(* Logix 5000 project; controller STAT 1756-L72 rev 20.12; software revision 20.04; part 24 of 34 *)
(* tags used below, declared in another part *)
   B3 : DINT[35];
   N9 : DINT[200];
   S : INT[164];
   T4 : TIMER[100];
   av310 : BOOL;
   av330 : BOOL;
   BITMW1 : BOOL;
   L4_R2_3_O : BOOL;
   S_AV310_V1_FC_C : BOOL;
   S_AV310_V1_FC_O : BOOL;
   S_AV310_V2_FC_C : BOOL;
   S_AV310_V2_FC_O : BOOL;
   S_AV330_V1_FC_C : BOOL;
   S_AV330_V1_FC_O : BOOL;
   S_AV330_V2_FC_C : BOOL;
   S_AV330_V2_FC_O : BOOL;
   stat_L1 : DINT[20];
   STAT_L3 : DINT[20];
(* LANCY, continued *)

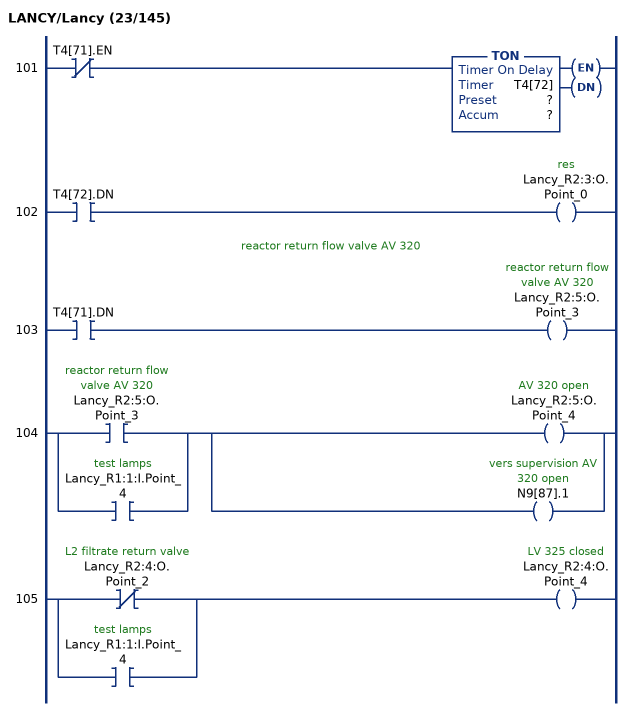
   101: XIO(T4[71].EN)TON(T4[72],?,?);
   102: XIC(T4[72].DN)OTE(Lancy_R2:3:O.Point_0);
   // reactor return flow valve AV 320
   103: XIC(T4[71].DN)OTE(Lancy_R2:5:O.Point_3);
   104: [XIC(Lancy_R2:5:O.Point_3) ,XIC(Lancy_R1:1:I.Point_4) ][OTE(Lancy_R2:5:O.Point_4) ,OTE(N9[87].1) ];
   105: [XIO(Lancy_R2:4:O.Point_2) ,XIC(Lancy_R1:1:I.Point_4) ]OTE(Lancy_R2:4:O.Point_4);
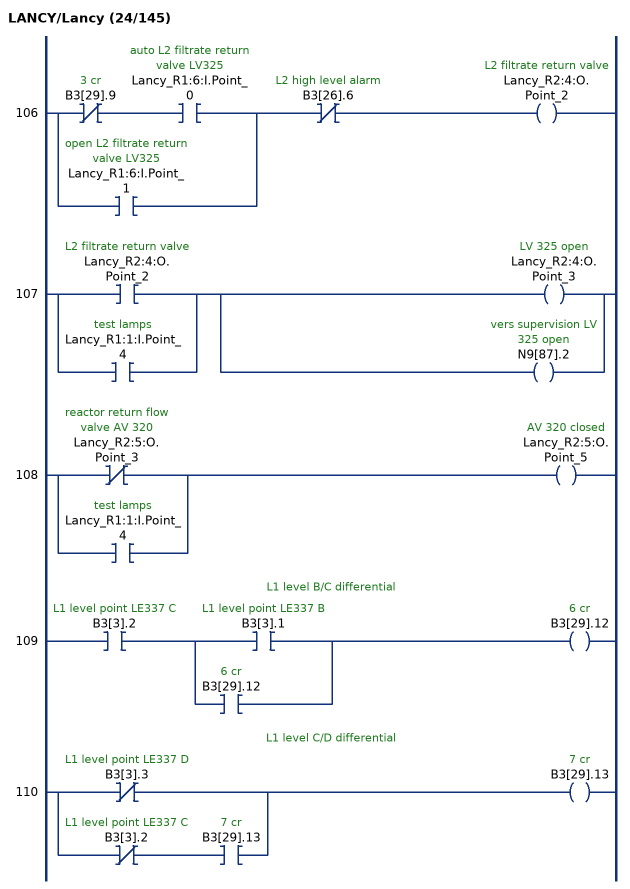
   106: [XIO(B3[29].9) XIC(Lancy_R1:6:I.Point_0) ,XIC(Lancy_R1:6:I.Point_1) ]XIO(B3[26].6)OTE(Lancy_R2:4:O.Point_2);
   107: [XIC(Lancy_R2:4:O.Point_2) ,XIC(Lancy_R1:1:I.Point_4) ][OTE(Lancy_R2:4:O.Point_3) ,OTE(N9[87].2) ];
   108: [XIO(Lancy_R2:5:O.Point_3) ,XIC(Lancy_R1:1:I.Point_4) ]OTE(Lancy_R2:5:O.Point_5);
   // L1 level B/C differential
   109: XIC(B3[3].2)[XIC(B3[3].1) ,XIC(B3[29].12) ]OTE(B3[29].12);
   // L1 level C/D differential
   110: [XIO(B3[3].3) ,XIO(B3[3].2) XIC(B3[29].13) ]OTE(B3[29].13);
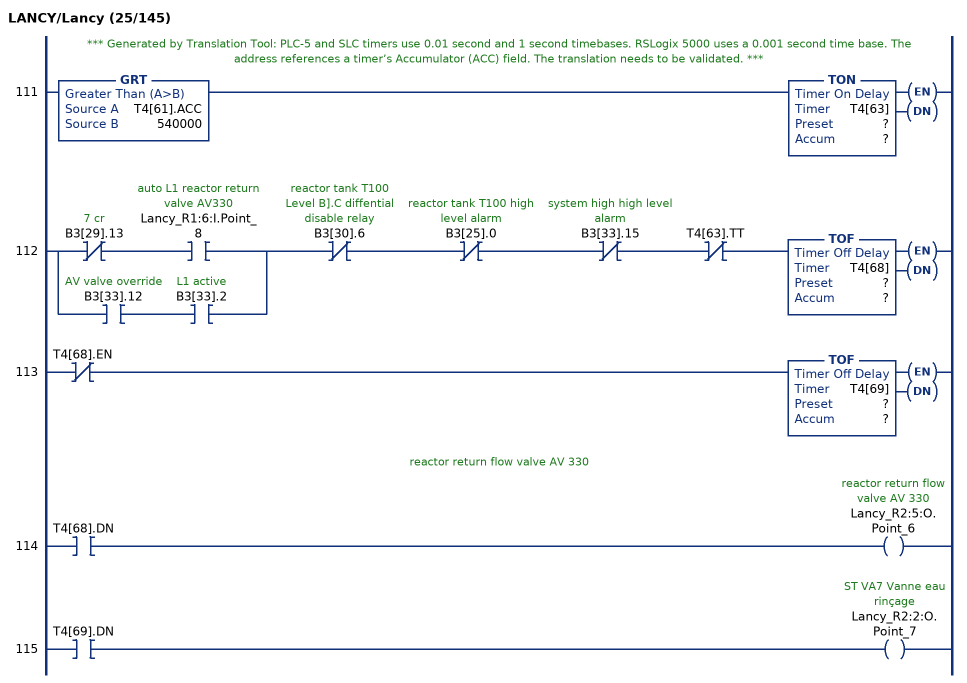
   // *** Generated by Translation Tool: PLC-5 and SLC timers use 0.01 second and 1 second timebases. RSLogix 5000 uses a 0.001 second time base. The address references a timer’s Accumulator (ACC) field. The translation needs to be validated. ***
   111: GRT(T4[61].ACC,540000)TON(T4[63],?,?);
   112: [XIO(B3[29].13) XIC(Lancy_R1:6:I.Point_8) ,XIC(B3[33].12) XIC(B3[33].2) ]XIO(B3[30].6)XIO(B3[25].0)XIO(B3[33].15)XIO(T4[63].TT)TOF(T4[68],?,?);
   113: XIO(T4[68].EN)TOF(T4[69],?,?);
   // reactor return flow valve AV 330
   114: XIC(T4[68].DN)OTE(Lancy_R2:5:O.Point_6);
   115: XIC(T4[69].DN)OTE(Lancy_R2:2:O.Point_7);
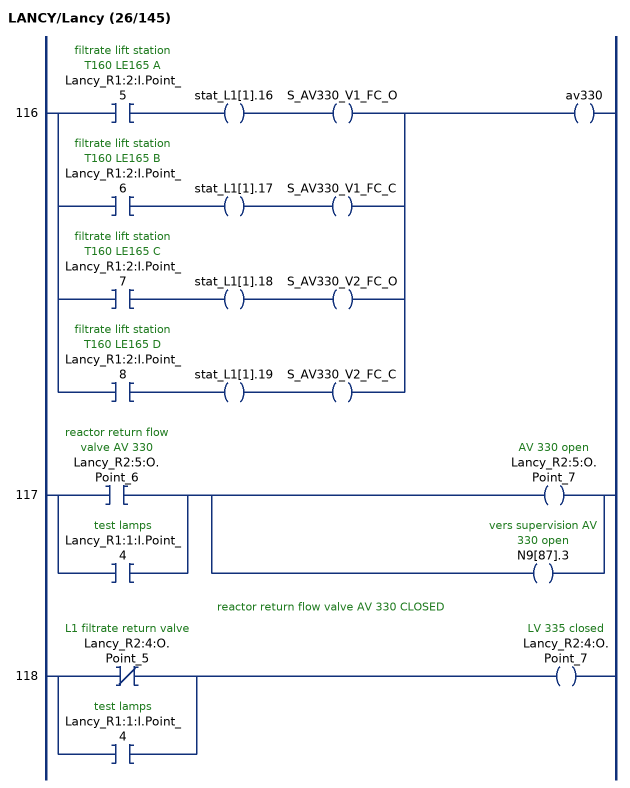
   116: [XIC(Lancy_R1:2:I.Point_5) OTE(stat_L1[1].16) OTE(S_AV330_V1_FC_O) ,XIC(Lancy_R1:2:I.Point_6) OTE(stat_L1[1].17) OTE(S_AV330_V1_FC_C) ,XIC(Lancy_R1:2:I.Point_7) OTE(stat_L1[1].18) OTE(S_AV330_V2_FC_O) ,XIC(Lancy_R1:2:I.Point_8) OTE(stat_L1[1].19) OTE(S_AV330_V2_FC_C) ]OTE(av330);
   117: [XIC(Lancy_R2:5:O.Point_6) ,XIC(Lancy_R1:1:I.Point_4) ][OTE(Lancy_R2:5:O.Point_7) ,OTE(N9[87].3) ];
   // reactor return flow valve AV 330 CLOSED
   118: [XIO(Lancy_R2:4:O.Point_5) ,XIC(Lancy_R1:1:I.Point_4) ]OTE(Lancy_R2:4:O.Point_7);
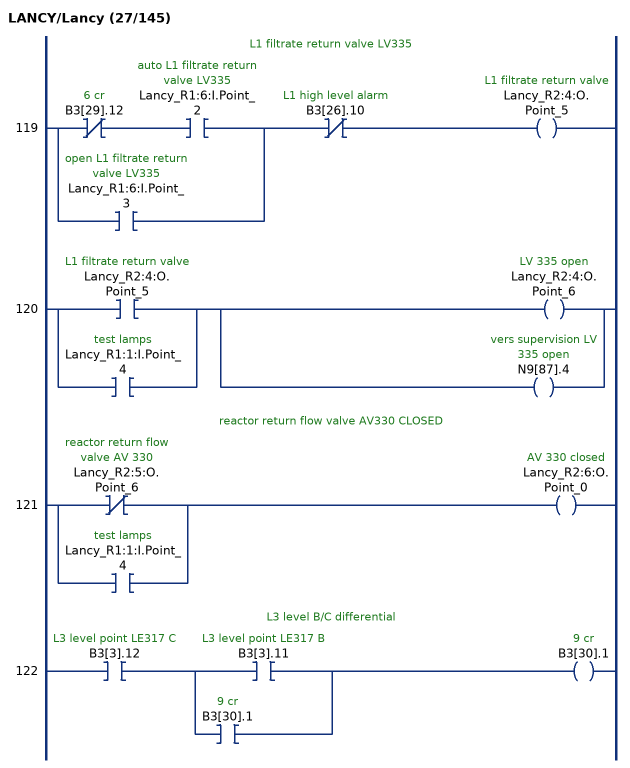
   // L1 filtrate return valve LV335
   119: [XIO(B3[29].12) XIC(Lancy_R1:6:I.Point_2) ,XIC(Lancy_R1:6:I.Point_3) ]XIO(B3[26].10)OTE(Lancy_R2:4:O.Point_5);
   120: [XIC(Lancy_R2:4:O.Point_5) ,XIC(Lancy_R1:1:I.Point_4) ][OTE(Lancy_R2:4:O.Point_6) ,OTE(N9[87].4) ];
   // reactor return flow valve AV330 CLOSED
   121: [XIO(Lancy_R2:5:O.Point_6) ,XIC(Lancy_R1:1:I.Point_4) ]OTE(Lancy_R2:6:O.Point_0);
   // L3 level B/C differential
   122: XIC(B3[3].12)[XIC(B3[3].11) ,XIC(B3[30].1) ]OTE(B3[30].1);
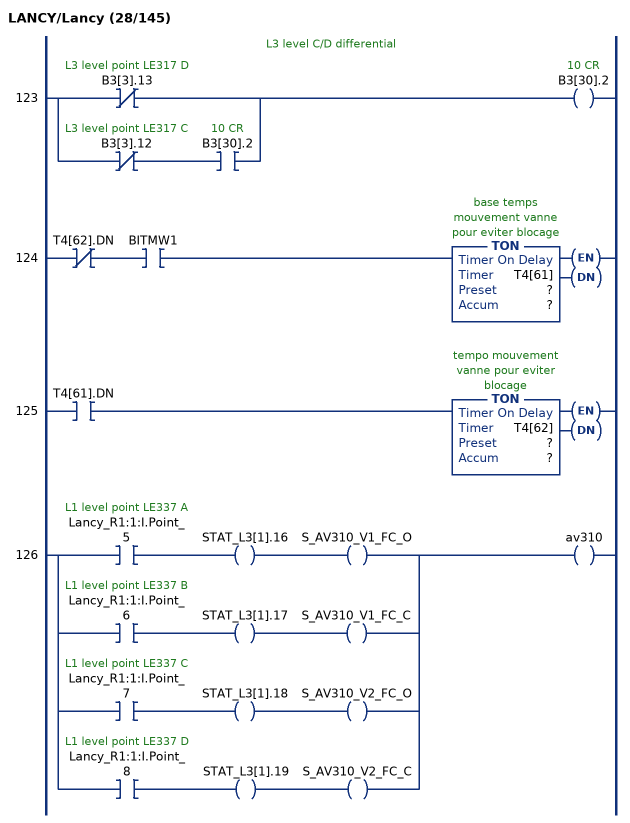
   // L3 level C/D differential
   123: [XIO(B3[3].13) ,XIO(B3[3].12) XIC(B3[30].2) ]OTE(B3[30].2);
   124: XIO(T4[62].DN)XIC(BITMW1)TON(T4[61],?,?);
   125: XIC(T4[61].DN)TON(T4[62],?,?);
   126: [XIC(Lancy_R1:1:I.Point_5) OTE(STAT_L3[1].16) OTE(S_AV310_V1_FC_O) ,XIC(Lancy_R1:1:I.Point_6) OTE(STAT_L3[1].17) OTE(S_AV310_V1_FC_C) ,XIC(Lancy_R1:1:I.Point_7) OTE(STAT_L3[1].18) OTE(S_AV310_V2_FC_O) ,XIC(Lancy_R1:1:I.Point_8) OTE(STAT_L3[1].19) OTE(S_AV310_V2_FC_C) ]OTE(av310);
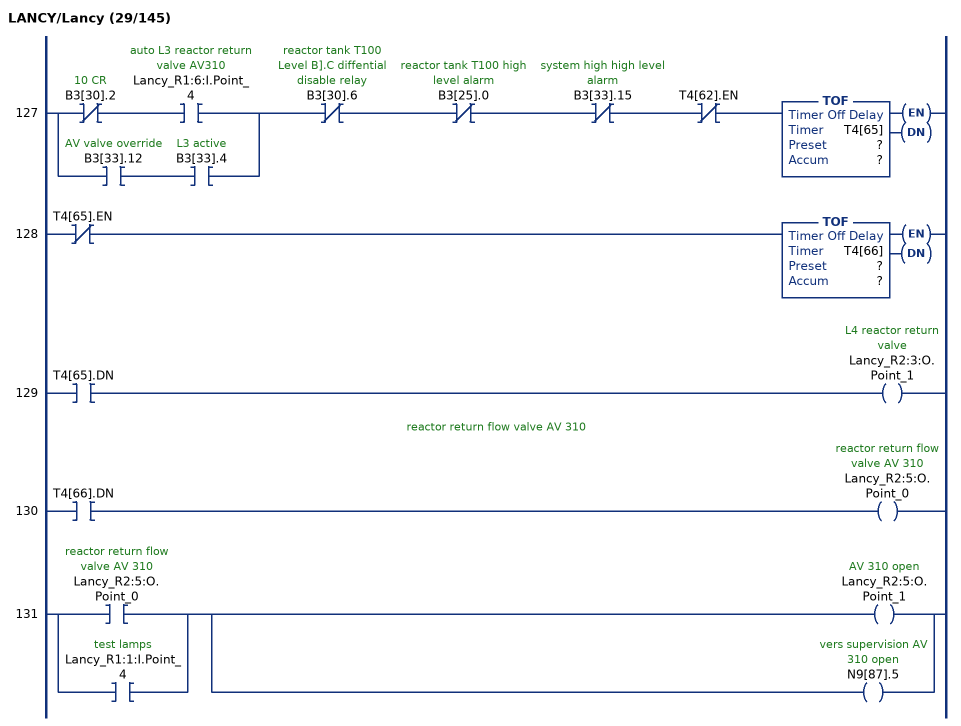
   127: [XIO(B3[30].2) XIC(Lancy_R1:6:I.Point_4) ,XIC(B3[33].12) XIC(B3[33].4) ]XIO(B3[30].6)XIO(B3[25].0)XIO(B3[33].15)XIO(T4[62].EN)TOF(T4[65],?,?);
   128: XIO(T4[65].EN)TOF(T4[66],?,?);
   129: XIC(T4[65].DN)OTE(Lancy_R2:3:O.Point_1);
   // reactor return flow valve AV 310
   130: XIC(T4[66].DN)OTE(Lancy_R2:5:O.Point_0);
   131: [XIC(Lancy_R2:5:O.Point_0) ,XIC(Lancy_R1:1:I.Point_4) ][OTE(Lancy_R2:5:O.Point_1) ,OTE(N9[87].5) ];
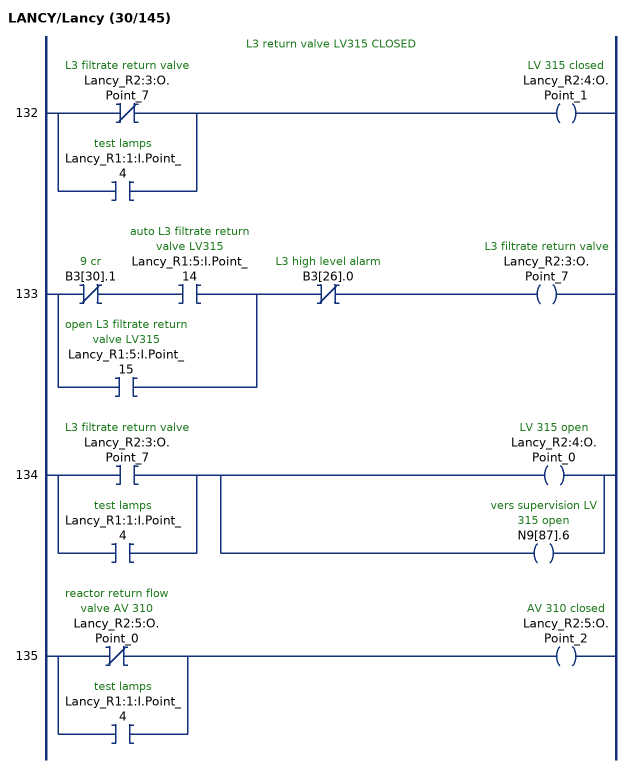
   // L3 return valve LV315 CLOSED
   132: [XIO(Lancy_R2:3:O.Point_7) ,XIC(Lancy_R1:1:I.Point_4) ]OTE(Lancy_R2:4:O.Point_1);
   133: [XIO(B3[30].1) XIC(Lancy_R1:5:I.Point_14) ,XIC(Lancy_R1:5:I.Point_15) ]XIO(B3[26].0)OTE(Lancy_R2:3:O.Point_7);
   134: [XIC(Lancy_R2:3:O.Point_7) ,XIC(Lancy_R1:1:I.Point_4) ][OTE(Lancy_R2:4:O.Point_0) ,OTE(N9[87].6) ];
   135: [XIO(Lancy_R2:5:O.Point_0) ,XIC(Lancy_R1:1:I.Point_4) ]OTE(Lancy_R2:5:O.Point_2);
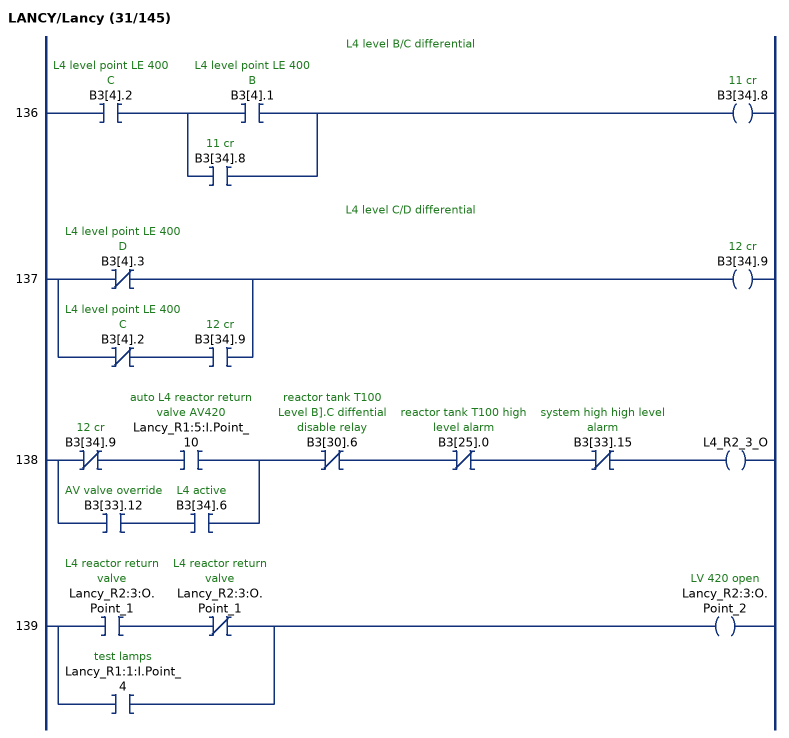
   // L4 level B/C differential
   136: XIC(B3[4].2)[XIC(B3[4].1) ,XIC(B3[34].8) ]OTE(B3[34].8);
   // L4 level C/D differential
   137: [XIO(B3[4].3) ,XIO(B3[4].2) XIC(B3[34].9) ]OTE(B3[34].9);
   138: [XIO(B3[34].9) XIC(Lancy_R1:5:I.Point_10) ,XIC(B3[33].12) XIC(B3[34].6) ]XIO(B3[30].6)XIO(B3[25].0)XIO(B3[33].15)OTE(L4_R2_3_O);
   139: [XIC(Lancy_R2:3:O.Point_1) XIO(Lancy_R2:3:O.Point_1) ,XIC(Lancy_R1:1:I.Point_4) ]OTE(Lancy_R2:3:O.Point_2);
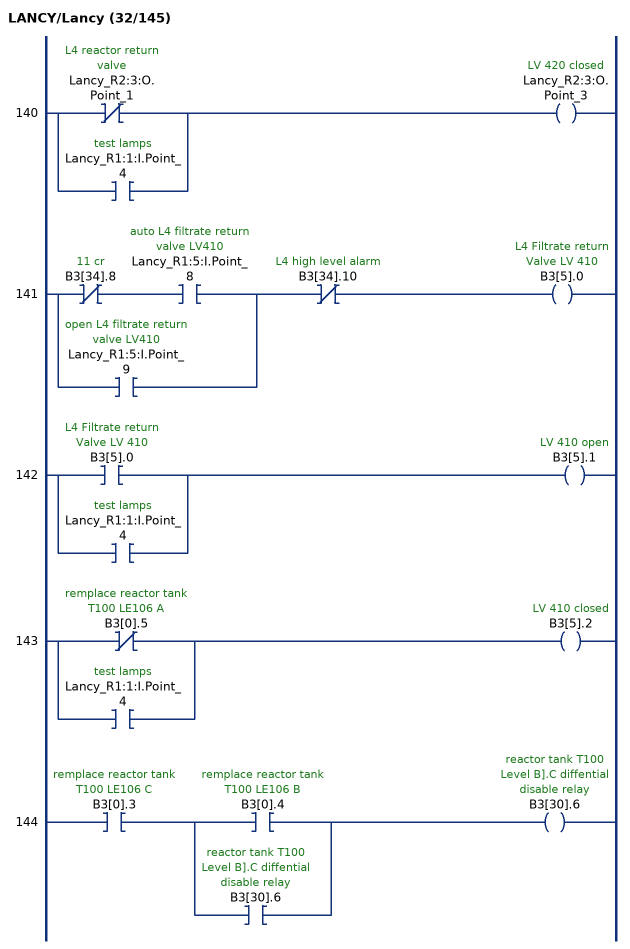
   140: [XIO(Lancy_R2:3:O.Point_1) ,XIC(Lancy_R1:1:I.Point_4) ]OTE(Lancy_R2:3:O.Point_3);
   141: [XIO(B3[34].8) XIC(Lancy_R1:5:I.Point_8) ,XIC(Lancy_R1:5:I.Point_9) ]XIO(B3[34].10)OTE(B3[5].0);
   142: [XIC(B3[5].0) ,XIC(Lancy_R1:1:I.Point_4) ]OTE(B3[5].1);
   143: [XIO(B3[0].5) ,XIC(Lancy_R1:1:I.Point_4) ]OTE(B3[5].2);
   144: XIC(B3[0].3)[XIC(B3[0].4) ,XIC(B3[30].6) ]OTE(B3[30].6);
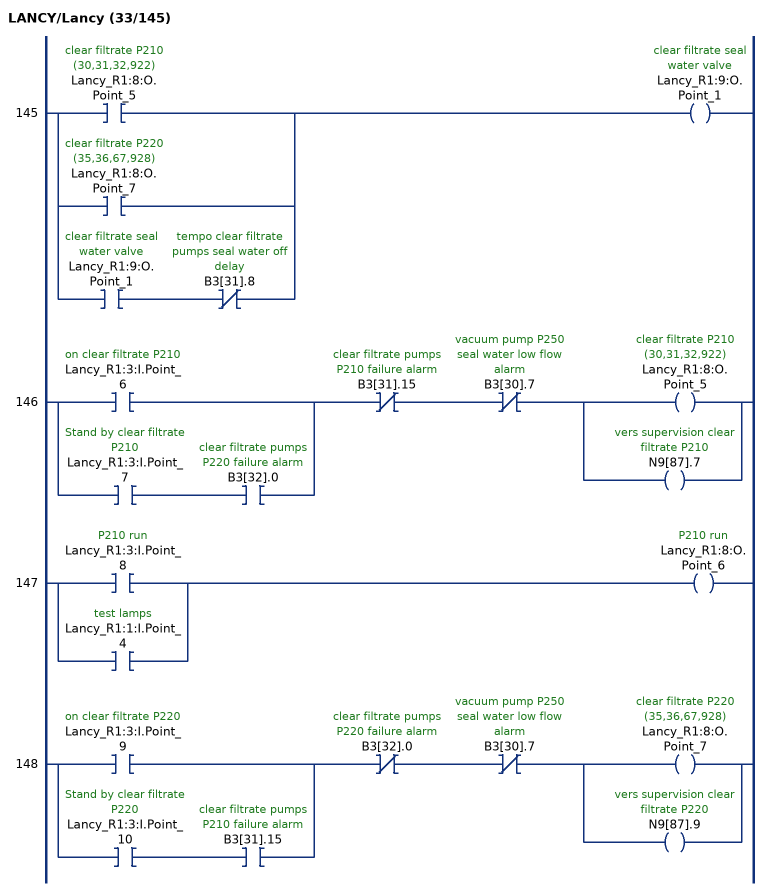
   145: [[XIC(Lancy_R1:8:O.Point_5) ,XIC(Lancy_R1:8:O.Point_7) ] ,XIC(Lancy_R1:9:O.Point_1) XIO(B3[31].8) ]OTE(Lancy_R1:9:O.Point_1);
   146: [XIC(Lancy_R1:3:I.Point_6) ,XIC(Lancy_R1:3:I.Point_7) XIC(B3[32].0) ]XIO(B3[31].15)XIO(B3[30].7)[OTE(Lancy_R1:8:O.Point_5) ,OTE(N9[87].7) ];
   147: [XIC(Lancy_R1:3:I.Point_8) ,XIC(Lancy_R1:1:I.Point_4) ]OTE(Lancy_R1:8:O.Point_6);
   148: [XIC(Lancy_R1:3:I.Point_9) ,XIC(Lancy_R1:3:I.Point_10) XIC(B3[31].15) ]XIO(B3[32].0)XIO(B3[30].7)[OTE(Lancy_R1:8:O.Point_7) ,OTE(N9[87].9) ];
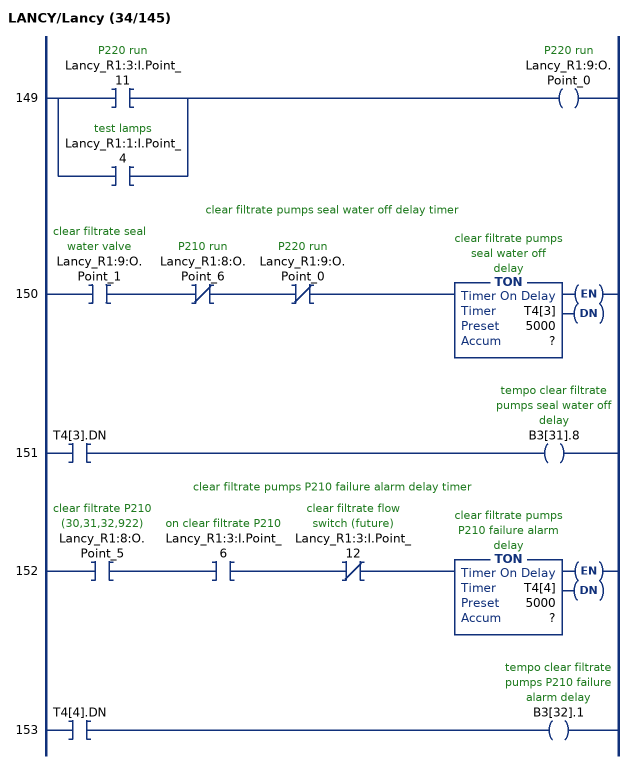
   149: [XIC(Lancy_R1:3:I.Point_11) ,XIC(Lancy_R1:1:I.Point_4) ]OTE(Lancy_R1:9:O.Point_0);
   // clear filtrate pumps seal water off delay timer
   150: XIC(Lancy_R1:9:O.Point_1)XIO(Lancy_R1:8:O.Point_6)XIO(Lancy_R1:9:O.Point_0)TON(T4[3],?,?);
   151: XIC(T4[3].DN)OTE(B3[31].8);
   // clear filtrate pumps P210 failure alarm delay timer
   152: XIC(Lancy_R1:8:O.Point_5)XIC(Lancy_R1:3:I.Point_6)XIO(Lancy_R1:3:I.Point_12)TON(T4[4],?,?);
   153: XIC(T4[4].DN)OTE(B3[32].1);
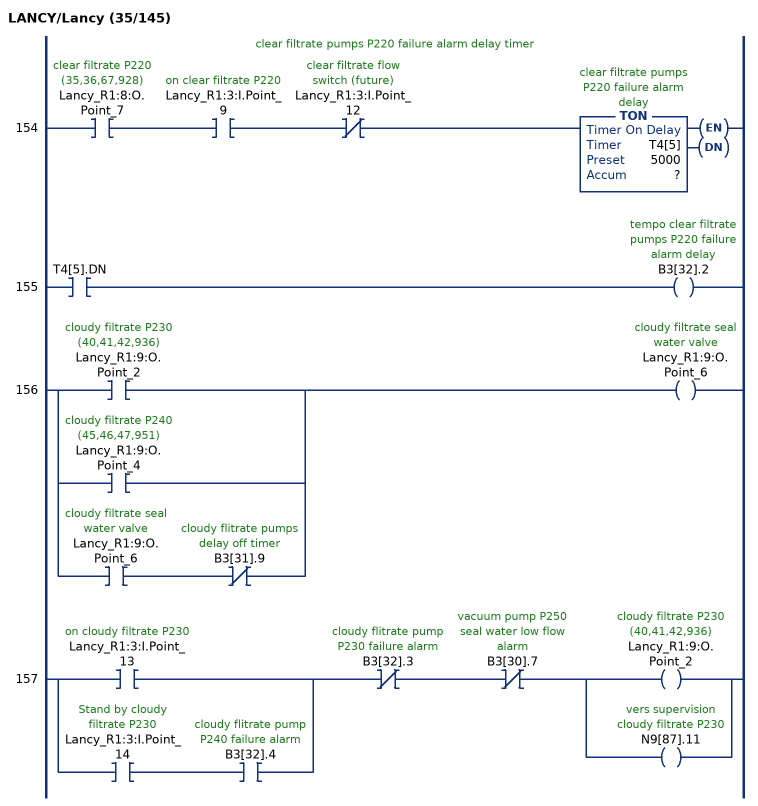
   // clear filtrate pumps P220 failure alarm delay timer
   154: XIC(Lancy_R1:8:O.Point_7)XIC(Lancy_R1:3:I.Point_9)XIO(Lancy_R1:3:I.Point_12)TON(T4[5],?,?);
   155: XIC(T4[5].DN)OTE(B3[32].2);
   156: [[XIC(Lancy_R1:9:O.Point_2) ,XIC(Lancy_R1:9:O.Point_4) ] ,XIC(Lancy_R1:9:O.Point_6) XIO(B3[31].9) ]OTE(Lancy_R1:9:O.Point_6);
   157: [XIC(Lancy_R1:3:I.Point_13) ,XIC(Lancy_R1:3:I.Point_14) XIC(B3[32].4) ]XIO(B3[32].3)XIO(B3[30].7)[OTE(Lancy_R1:9:O.Point_2) ,OTE(N9[87].11) ];
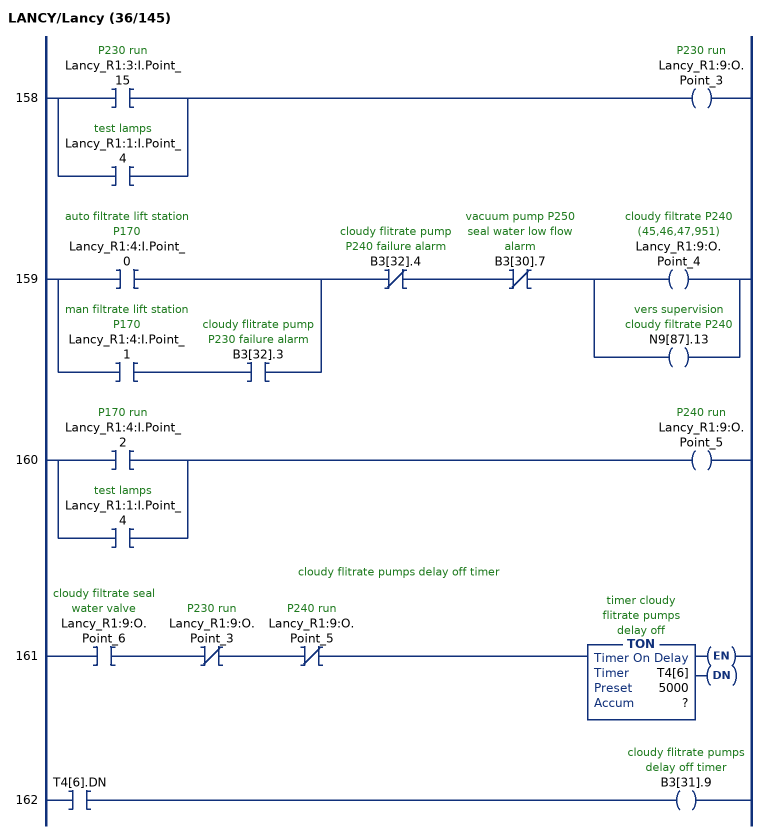
   158: [XIC(Lancy_R1:3:I.Point_15) ,XIC(Lancy_R1:1:I.Point_4) ]OTE(Lancy_R1:9:O.Point_3);
   159: [XIC(Lancy_R1:4:I.Point_0) ,XIC(Lancy_R1:4:I.Point_1) XIC(B3[32].3) ]XIO(B3[32].4)XIO(B3[30].7)[OTE(Lancy_R1:9:O.Point_4) ,OTE(N9[87].13) ];
   160: [XIC(Lancy_R1:4:I.Point_2) ,XIC(Lancy_R1:1:I.Point_4) ]OTE(Lancy_R1:9:O.Point_5);
   // cloudy flitrate pumps delay off timer
   161: XIC(Lancy_R1:9:O.Point_6)XIO(Lancy_R1:9:O.Point_3)XIO(Lancy_R1:9:O.Point_5)TON(T4[6],?,?);
   162: XIC(T4[6].DN)OTE(B3[31].9);
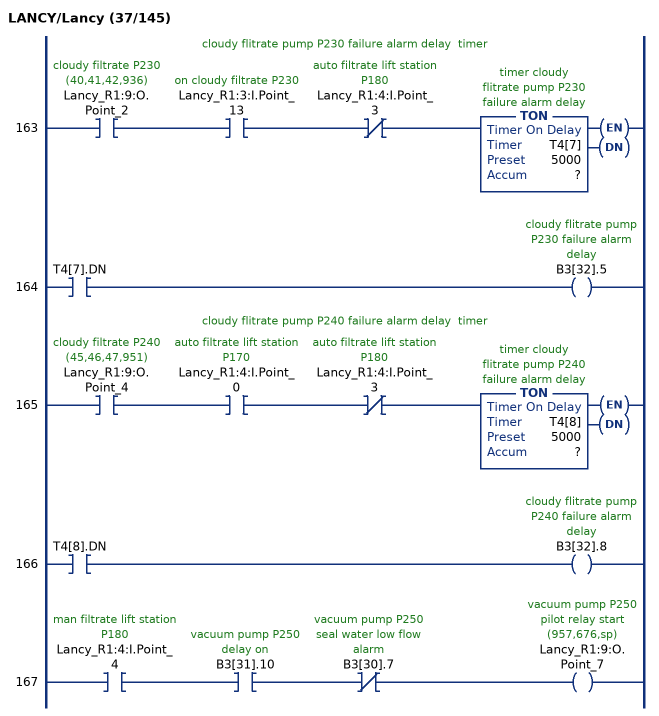
   // cloudy flitrate pump P230 failure alarm delay  timer
   163: XIC(Lancy_R1:9:O.Point_2)XIC(Lancy_R1:3:I.Point_13)XIO(Lancy_R1:4:I.Point_3)TON(T4[7],?,?);
   164: XIC(T4[7].DN)OTE(B3[32].5);
   // cloudy flitrate pump P240 failure alarm delay  timer
   165: XIC(Lancy_R1:9:O.Point_4)XIC(Lancy_R1:4:I.Point_0)XIO(Lancy_R1:4:I.Point_3)TON(T4[8],?,?);
   166: XIC(T4[8].DN)OTE(B3[32].8);
   167: XIC(Lancy_R1:4:I.Point_4)XIC(B3[31].10)XIO(B3[30].7)OTE(Lancy_R1:9:O.Point_7);
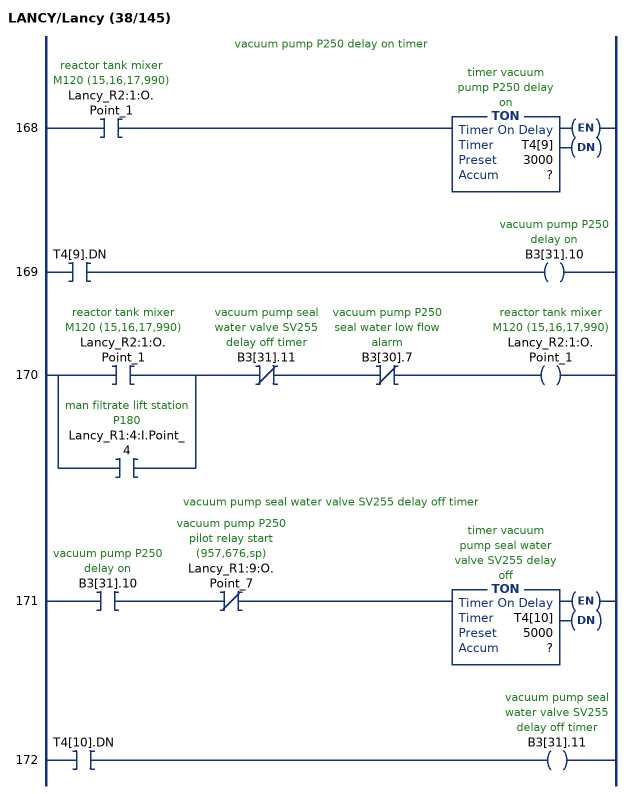
   // vacuum pump P250 delay on timer
   168: XIC(Lancy_R2:1:O.Point_1)TON(T4[9],?,?);
   169: XIC(T4[9].DN)OTE(B3[31].10);
   170: [XIC(Lancy_R2:1:O.Point_1) ,XIC(Lancy_R1:4:I.Point_4) ]XIO(B3[31].11)XIO(B3[30].7)OTE(Lancy_R2:1:O.Point_1);
   // vacuum pump seal water valve SV255 delay off timer
   171: XIC(B3[31].10)XIO(Lancy_R1:9:O.Point_7)TON(T4[10],?,?);
   172: XIC(T4[10].DN)OTE(B3[31].11);
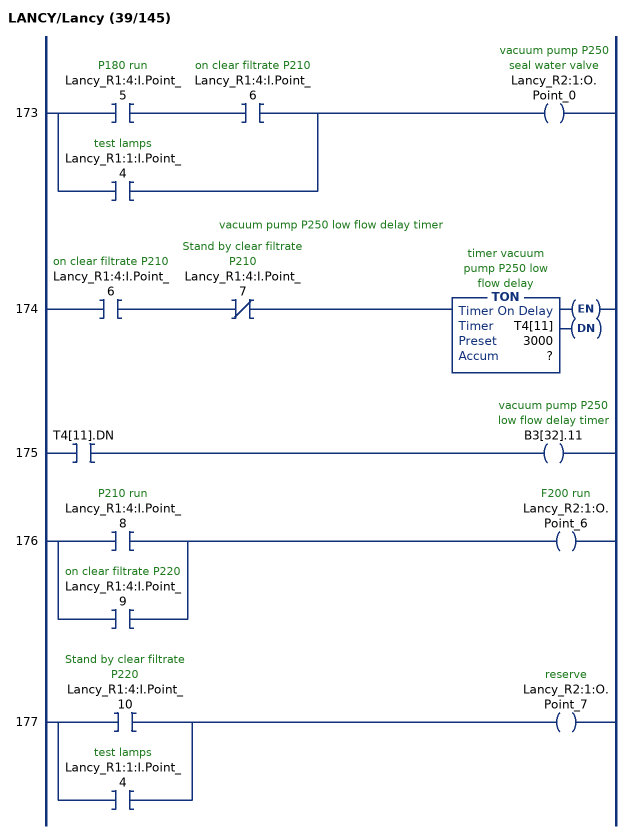
   173: [XIC(Lancy_R1:4:I.Point_5) XIC(Lancy_R1:4:I.Point_6) ,XIC(Lancy_R1:1:I.Point_4) ]OTE(Lancy_R2:1:O.Point_0);
   // vacuum pump P250 low flow delay timer
   174: XIC(Lancy_R1:4:I.Point_6)XIO(Lancy_R1:4:I.Point_7)TON(T4[11],?,?);
   175: XIC(T4[11].DN)OTE(B3[32].11);
   176: [XIC(Lancy_R1:4:I.Point_8) ,XIC(Lancy_R1:4:I.Point_9) ]OTE(Lancy_R2:1:O.Point_6);
   177: [XIC(Lancy_R1:4:I.Point_10) ,XIC(Lancy_R1:1:I.Point_4) ]OTE(Lancy_R2:1:O.Point_7);
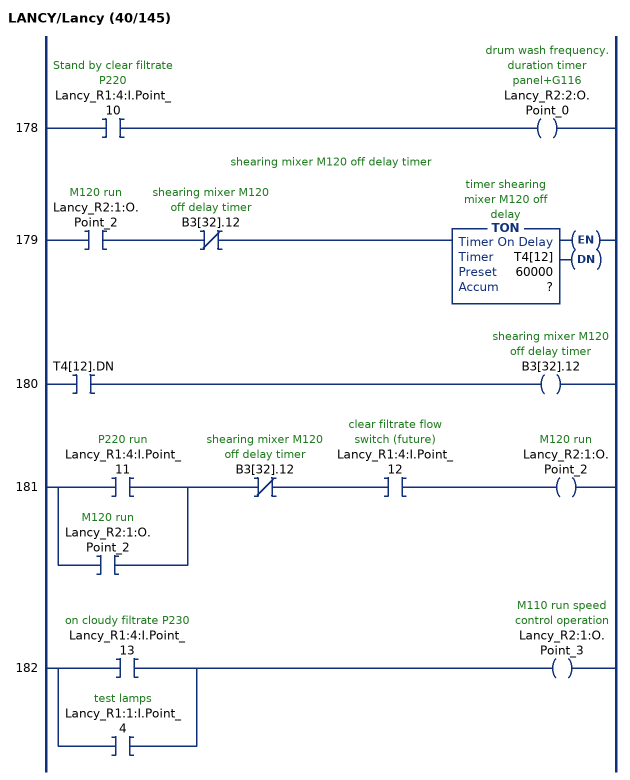
   178: XIC(Lancy_R1:4:I.Point_10)OTE(Lancy_R2:2:O.Point_0);
   // shearing mixer M120 off delay timer
   179: XIC(Lancy_R2:1:O.Point_2)XIO(B3[32].12)TON(T4[12],?,?);
   180: XIC(T4[12].DN)OTE(B3[32].12);
   181: [XIC(Lancy_R1:4:I.Point_11) ,XIC(Lancy_R2:1:O.Point_2) ]XIO(B3[32].12)XIC(Lancy_R1:4:I.Point_12)OTE(Lancy_R2:1:O.Point_2);
   182: [XIC(Lancy_R1:4:I.Point_13) ,XIC(Lancy_R1:1:I.Point_4) ]OTE(Lancy_R2:1:O.Point_3);
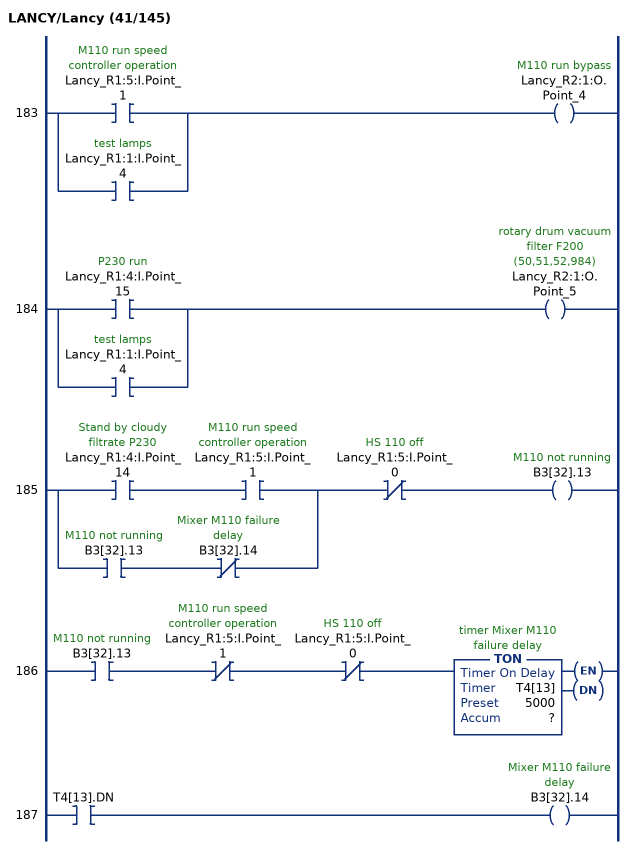
   183: [XIC(Lancy_R1:5:I.Point_1) ,XIC(Lancy_R1:1:I.Point_4) ]OTE(Lancy_R2:1:O.Point_4);
   184: [XIC(Lancy_R1:4:I.Point_15) ,XIC(Lancy_R1:1:I.Point_4) ]OTE(Lancy_R2:1:O.Point_5);
   185: [XIC(Lancy_R1:4:I.Point_14) XIC(Lancy_R1:5:I.Point_1) ,XIC(B3[32].13) XIO(B3[32].14) ]XIO(Lancy_R1:5:I.Point_0)OTE(B3[32].13);
   186: XIC(B3[32].13)XIO(Lancy_R1:5:I.Point_1)XIO(Lancy_R1:5:I.Point_0)TON(T4[13],?,?);
   187: XIC(T4[13].DN)OTE(B3[32].14);
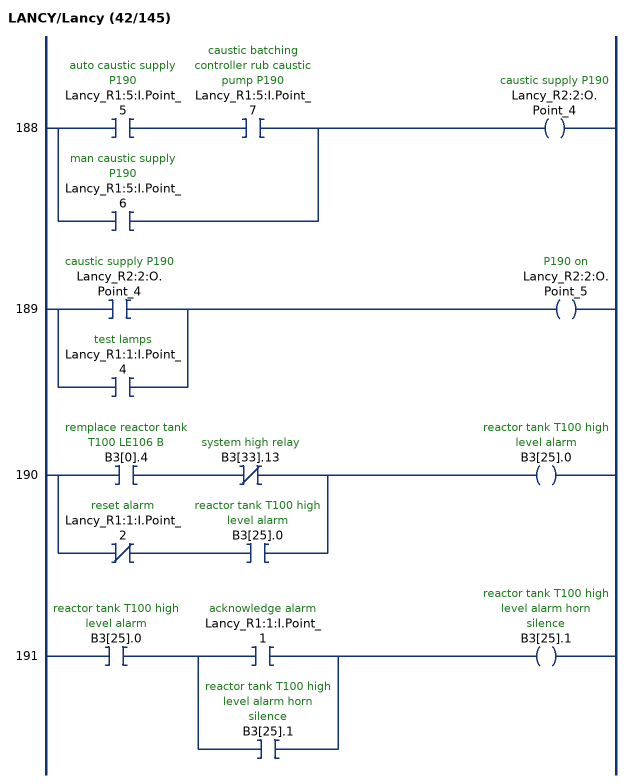
   188: [XIC(Lancy_R1:5:I.Point_5) XIC(Lancy_R1:5:I.Point_7) ,XIC(Lancy_R1:5:I.Point_6) ]OTE(Lancy_R2:2:O.Point_4);
   189: [XIC(Lancy_R2:2:O.Point_4) ,XIC(Lancy_R1:1:I.Point_4) ]OTE(Lancy_R2:2:O.Point_5);
   190: [XIC(B3[0].4) XIO(B3[33].13) ,XIO(Lancy_R1:1:I.Point_2) XIC(B3[25].0) ]OTE(B3[25].0);
   191: XIC(B3[25].0)[XIC(Lancy_R1:1:I.Point_1) ,XIC(B3[25].1) ]OTE(B3[25].1);
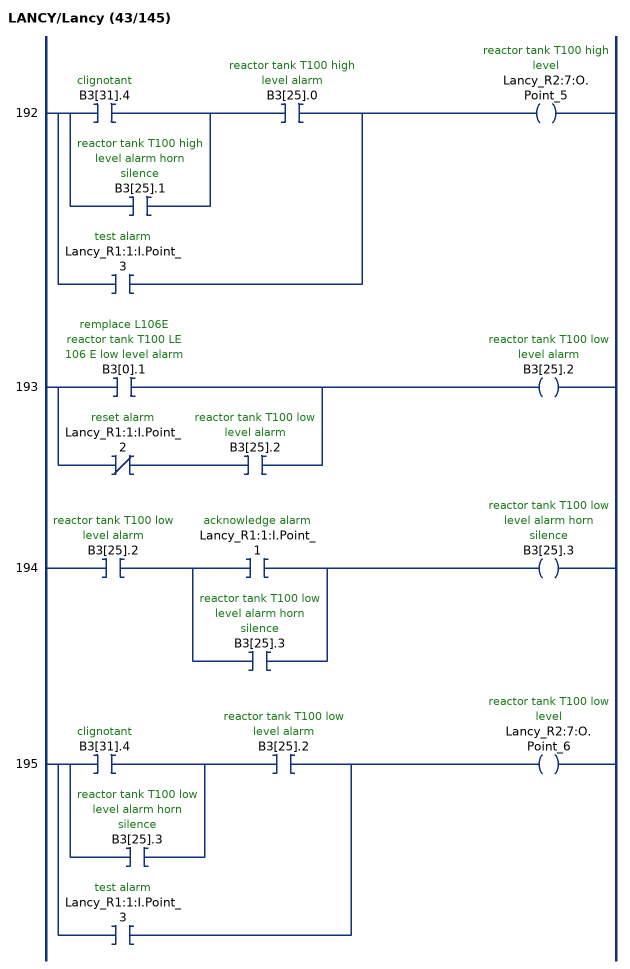
   192: [[XIC(B3[31].4) ,XIC(B3[25].1) ] XIC(B3[25].0) ,XIC(Lancy_R1:1:I.Point_3) ]OTE(Lancy_R2:7:O.Point_5);
   193: [XIC(B3[0].1) ,XIO(Lancy_R1:1:I.Point_2) XIC(B3[25].2) ]OTE(B3[25].2);
   194: XIC(B3[25].2)[XIC(Lancy_R1:1:I.Point_1) ,XIC(B3[25].3) ]OTE(B3[25].3);
   195: [[XIC(B3[31].4) ,XIC(B3[25].3) ] XIC(B3[25].2) ,XIC(Lancy_R1:1:I.Point_3) ]OTE(Lancy_R2:7:O.Point_6);
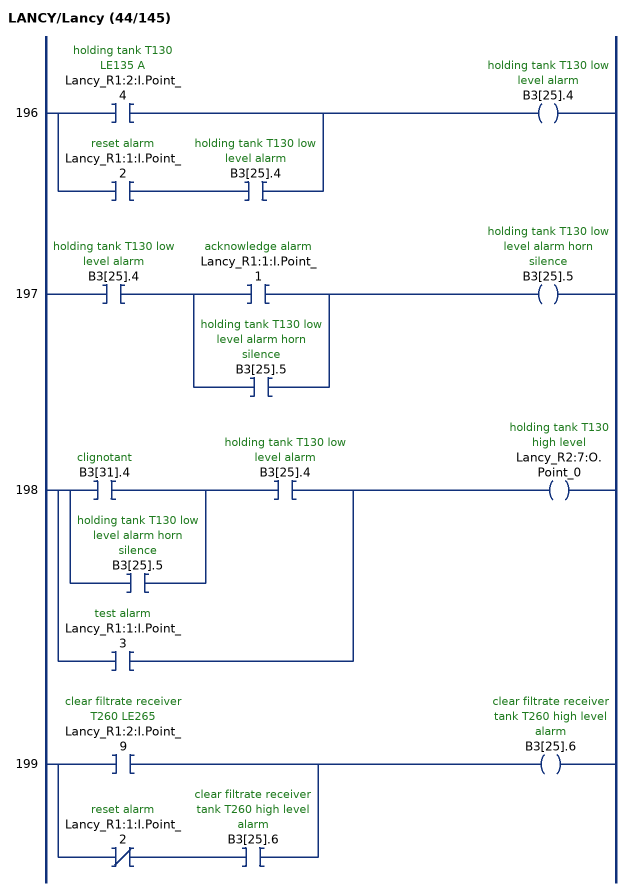
   196: [XIC(Lancy_R1:2:I.Point_4) ,XIC(Lancy_R1:1:I.Point_2) XIC(B3[25].4) ]OTE(B3[25].4);
   197: XIC(B3[25].4)[XIC(Lancy_R1:1:I.Point_1) ,XIC(B3[25].5) ]OTE(B3[25].5);
   198: [[XIC(B3[31].4) ,XIC(B3[25].5) ] XIC(B3[25].4) ,XIC(Lancy_R1:1:I.Point_3) ]OTE(Lancy_R2:7:O.Point_0);
   199: [XIC(Lancy_R1:2:I.Point_9) ,XIO(Lancy_R1:1:I.Point_2) XIC(B3[25].6) ]OTE(B3[25].6);
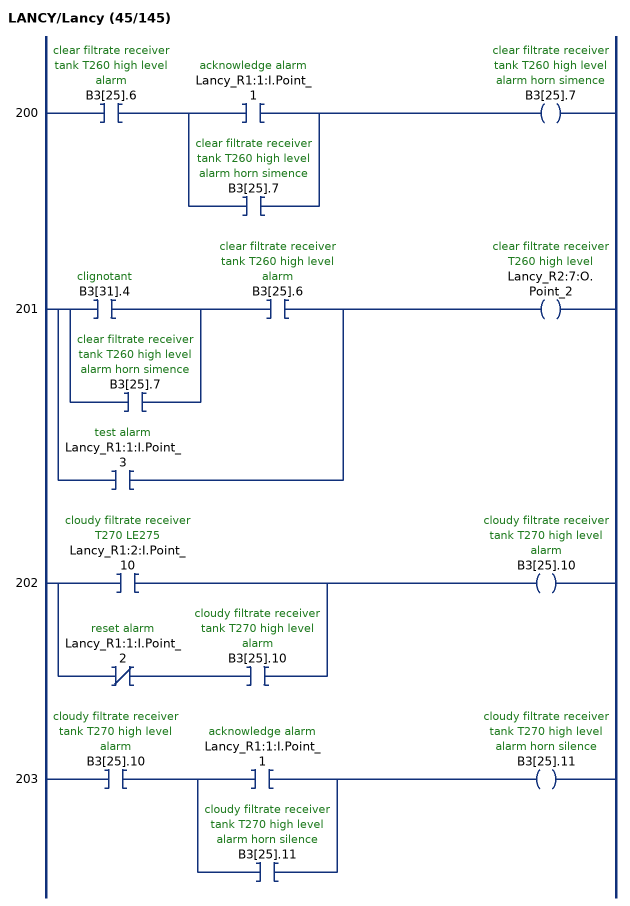
   200: XIC(B3[25].6)[XIC(Lancy_R1:1:I.Point_1) ,XIC(B3[25].7) ]OTE(B3[25].7);
   201: [[XIC(B3[31].4) ,XIC(B3[25].7) ] XIC(B3[25].6) ,XIC(Lancy_R1:1:I.Point_3) ]OTE(Lancy_R2:7:O.Point_2);
   202: [XIC(Lancy_R1:2:I.Point_10) ,XIO(Lancy_R1:1:I.Point_2) XIC(B3[25].10) ]OTE(B3[25].10);
   203: XIC(B3[25].10)[XIC(Lancy_R1:1:I.Point_1) ,XIC(B3[25].11) ]OTE(B3[25].11);
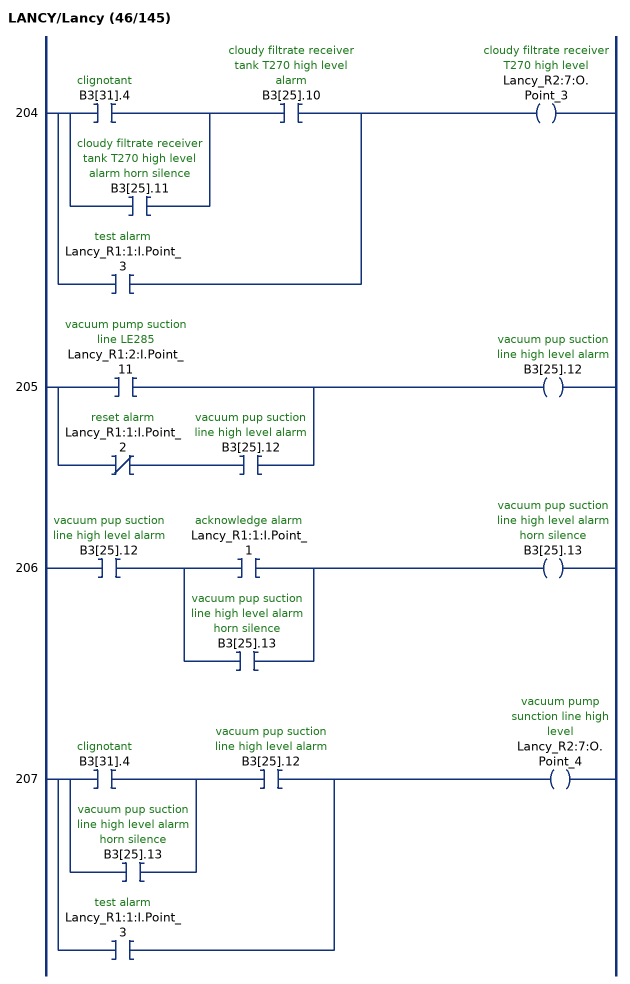
   204: [[XIC(B3[31].4) ,XIC(B3[25].11) ] XIC(B3[25].10) ,XIC(Lancy_R1:1:I.Point_3) ]OTE(Lancy_R2:7:O.Point_3);
   205: [XIC(Lancy_R1:2:I.Point_11) ,XIO(Lancy_R1:1:I.Point_2) XIC(B3[25].12) ]OTE(B3[25].12);
   206: XIC(B3[25].12)[XIC(Lancy_R1:1:I.Point_1) ,XIC(B3[25].13) ]OTE(B3[25].13);
   207: [[XIC(B3[31].4) ,XIC(B3[25].13) ] XIC(B3[25].12) ,XIC(Lancy_R1:1:I.Point_3) ]OTE(Lancy_R2:7:O.Point_4);
